PROGRAM EndurancePyrometerConstants
VAR CONSTANT
	ErrorCodes	: ST_EndurancePyrometerErrorCodes;
	Commands	: ST_EndurancePyrometerCommands;	
END_VAR

END_PROGRAM

(* stored: Version 1.1.0.1, ProductVersion 3.1.4024.16
   POU EndurancePyrometerConstants: Id {24835011-0abb-0638-39a8-d03c153a56cd}, SpecialFunc None *)
